PROGRAM OutDistributor
VAR
	bInput1 AT%I* : BOOL;
	bInput2 AT%I* : BOOL;
	bInput3 AT%I* : BOOL;
	bInput4 AT%I* : BOOL;
	bOutput AT%Q* : BOOL;
END_VAR

bOutput := bInput1 OR bInput2 OR bInput3 OR bInput4;

END_PROGRAM

(* stored: Version 1.1.0.1, ProductVersion 3.1.4024.6
   POU OutDistributor: Id {ae2aa4fe-42a2-4580-a91d-8284e35df4de}, SpecialFunc None *)
